(* Logix 5000 project; controller CIPDemo1 Emulate 5570 rev 32.11; software revision 32.00 *)

TASK MainTask (continuous, watchdog 500 ms) : MainProgram

MODULES
   Local : Emulate 5570 (ICP 3, rev 32.11)
END_MODULES

TYPE STR_3900 :   // <exclude/> Long string used in Big Dictionary
STRUCT
   LEN : DINT;
   DATA : SINT[3900];
END_STRUCT
END_TYPE

TYPE TXT_BIG_DICTIONARY :   // Big Dictionary used for storing and indexing strings.
STRUCT
   Index : TXT_DICTIONARY_INDEX[40000];   // Information to seek a text
   Items : STR_3900[414];
END_STRUCT
END_TYPE

TYPE TXT_DICTIONARY_INDEX :   // Index used in Big Dictionary
STRUCT
   Start : DINT;   // Start Index of text
   Size : INT;   // Actual Text Size
   Reserve : INT;   // Max reserved. 0=dynamic or not reserved
   PriorityGroup : INT;   // virtual grouping of dictionary entries OR Priority Number when used as message buffer
END_STRUCT
END_TYPE

VAR_GLOBAL   (* controller tags *)
   rate : DINT;
   tag1 : DINT;
   tag2 : REAL;
   text1 : STRING;
   TotalCount : DINT;
   TRK_Global_DictionaryWorkA : TXT_BIG_DICTIONARY;
END_VAR

PROGRAM MainProgram   (* main routine MainRoutine *)

ROUTINE MainRoutine   (* ladder *)
END_ROUTINE
END_PROGRAM
